Omron CX-Programmer project NewProject (CX-Programmer 9.75)

# PLC NewPLC1: CP2E-N N

## Global symbols (name address type ; comment)
0 CHANNEL  ; VIN1
0.00 BOOL  ; TIMER
0.01 BOOL  ; Auto
0.03 BOOL  ; Manual
1 CHANNEL  ; VIN1
100.01 BOOL  ; Tes
100.03 BOOL  ; 3C4
102 CHANNEL  ; INPUT 1 and 2 ACTIVE, AVERAGING, 0-10 V INPUT
103 CHANNEL  ; INPUT 3 AND 4 0-10V
2 CHANNEL  ; VIN1
3 CHANNEL  ; Potensiometer Input
4 CHANNEL  ; VIN3
5 CHANNEL  ; Timer every 500 ms mengambil data sensor
6 CHANNEL  ; VIN3
7 CHANNEL  ; VIN3
D0 CHANNEL  ; POTENTIOMETER
D1 CHANNEL  ; Panas
D10 CHANNEL  ; Parameter Sensor Suhu
D14 CHANNEL  ; Parameter Potentiometer
D151 CHANNEL  ; BIN to FLOAT Sensor Panas Multiply
D152 CHANNEL  ; Regression Multiply
D153 CHANNEL  ; Sensor Panas Float Unbiased
D154 CHANNEL  ; Bias Sensor Panas
D161 CHANNEL  ; Sensor Panas Float Unscaled
D170 CHANNEL  ; Bin to FLOAT Sensor division
D171 CHANNEL  ; BIN to FLOAT TRANSIMTTER DINGIN
D181 CHANNEL  ; Sensor Dingin Float Unscaled
D182 CHANNEL  ; Sensor Dingin Regression
D183 CHANNEL  ; Sensor Dingin no bias
D2 CHANNEL  ; Dingin
D20 CHANNEL  ; Hysterisis Input
D201 CHANNEL  ; DINGIN BIAS
D21 CHANNEL  ; Float Hysterisis Input
D30 CHANNEL  ; Scaled Sensor Dingin
D31 CHANNEL  ; Scaled Sensor Panas
D32 CHANNEL  ; Scaled Potentiometer FLOAT
D33 CHANNEL  ; Sensor Dingin Scaled
D34 CHANNEL  ; Scaled Sensor Panas
D35 CHANNEL  ; in bcd
D41 CHANNEL  ; Set atas
D42 CHANNEL  ; Set bawah
D70 CHANNEL  ; POTENTIOMETER FLOAT DIVIDER
D71 CHANNEL  ; POTENTIOMETER MULTIP FACTOR
D72 CHANNEL  ; POTENTIOMETER REGRESSION
D77 CHANNEL  ; POTENSIOMETER MULTIP FLOAT
D90 CHANNEL  ; UINT SENSOR DINGIN
D91 CHANNEL  ; UINT SENSOR PANAS
D92 CHANNEL  ; UINT POTENTIOMETER
T000 BOOL  ; TIMER
T001 BOOL  ; TIM2
LAMP 101.00 BOOL  ; Peltier
PELTIER 100.02 BOOL  ; 3C5
Switch 0.00 BOOL

## Program NewProgram1 (cyclic task 0)

### Section Initiation_and_Moving_Var

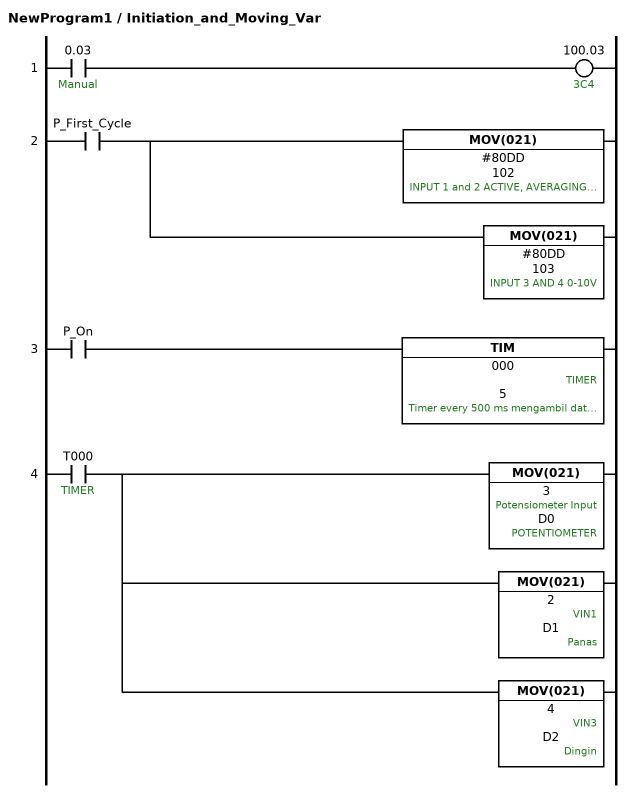
; rung 1
LD 0.03  ; Manual
OUT 100.03  ; 3C4
; rung 2
LD P_First_Cycle
MOV(021) #80DD 102  ; INPUT 1 and 2 ACTIVE, AVERAGING, 0-10 V INPUT
MOV(021) #80DD 103  ; INPUT 3 AND 4 0-10V
; rung 3
LD P_On
TIM 000 5  ; Timer every 500 ms mengambil data sensor, TIMER
; rung 4
LD T000  ; TIMER
MOV(021) 3 D0  ; Potensiometer Input, POTENTIOMETER
MOV(021) 2 D1  ; VIN1, Panas
MOV(021) 4 D2  ; VIN3, Dingin

### Section Scaling

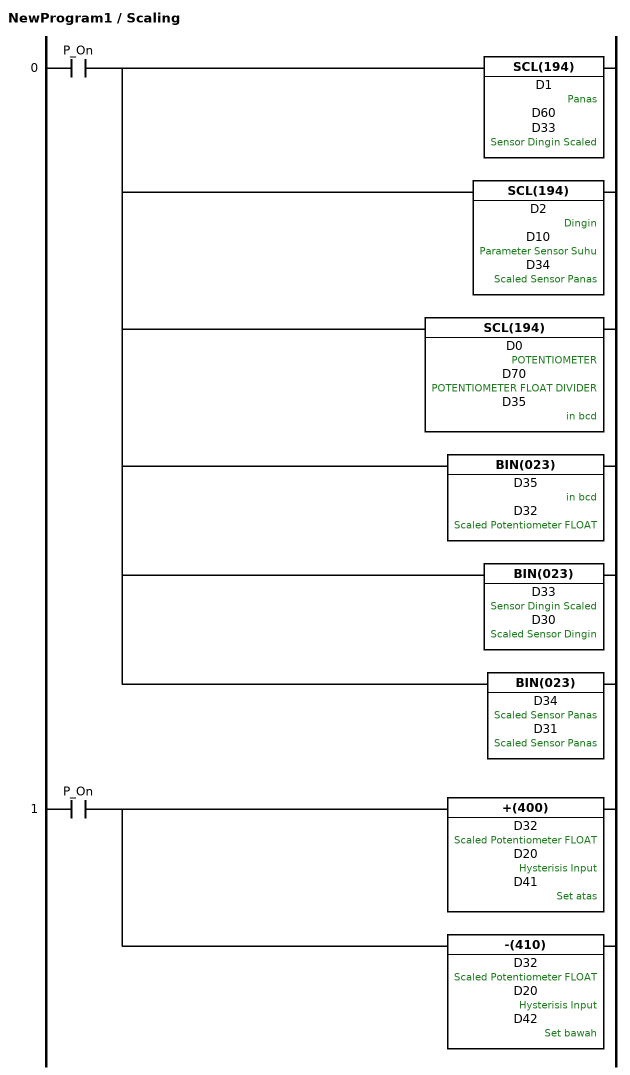
; rung 0
LD P_On
SCL(194) D1 D60 D33  ; Panas, Sensor Dingin Scaled
SCL(194) D2 D10 D34  ; Dingin, Parameter Sensor Suhu, Scaled Sensor Panas
SCL(194) D0 D70 D35  ; POTENTIOMETER, POTENTIOMETER FLOAT DIVIDER, in bcd
BIN(023) D35 D32  ; in bcd, Scaled Potentiometer FLOAT
BIN(023) D33 D30  ; Sensor Dingin Scaled, Scaled Sensor Dingin
BIN(023) D34 D31  ; Scaled Sensor Panas
; rung 1
LD P_On
+(400) D32 D20 D41  ; Scaled Potentiometer FLOAT, Hysterisis Input, Set atas
-(410) D32 D20 D42  ; Scaled Potentiometer FLOAT, Hysterisis Input, Set bawah

### Section Control

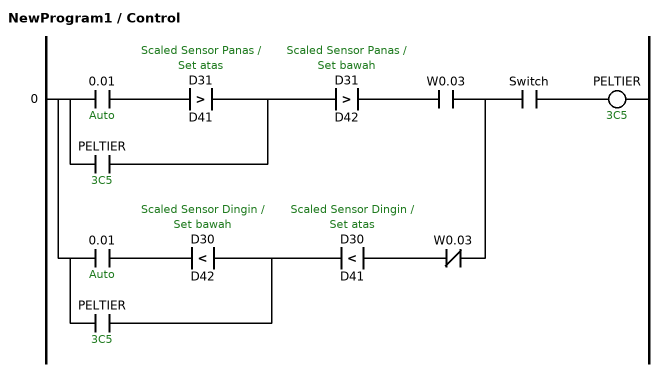
; rung 0
LD 0.01  ; Auto
AND>(320) D31 D41  ; Scaled Sensor Panas, Set atas
OR PELTIER  ; 3C5
AND>(320) D31 D42  ; Scaled Sensor Panas, Set bawah
AND W0.03
LD 0.01  ; Auto
AND<(310) D30 D42  ; Scaled Sensor Dingin, Set bawah
OR PELTIER  ; 3C5
AND<(310) D30 D41  ; Scaled Sensor Dingin, Set atas
ANDNOT W0.03
ORLD
AND Switch
OUT PELTIER  ; 3C5

### Section nyimpen

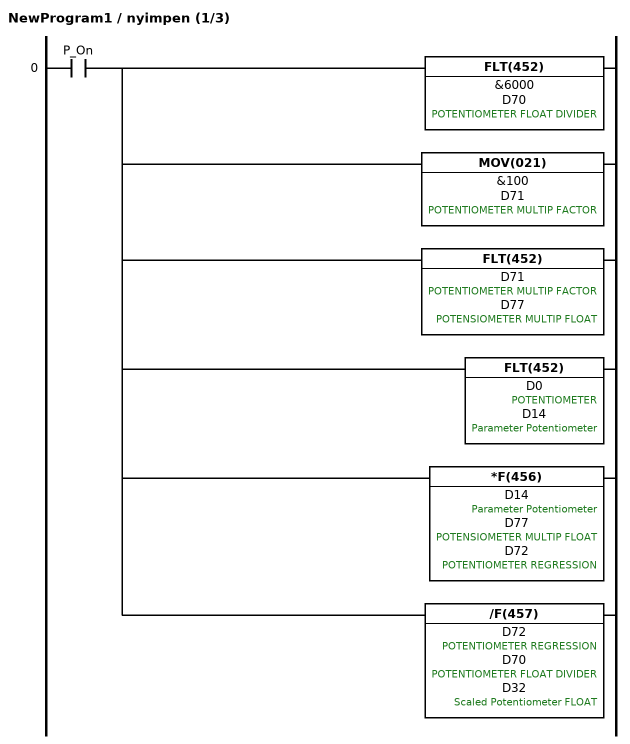
; rung 0
LD P_On
FLT(452) &6000 D70  ; POTENTIOMETER FLOAT DIVIDER
MOV(021) &100 D71  ; POTENTIOMETER MULTIP FACTOR
FLT(452) D71 D77  ; POTENTIOMETER MULTIP FACTOR, POTENSIOMETER MULTIP FLOAT
FLT(452) D0 D14  ; POTENTIOMETER, Parameter Potentiometer
*F(456) D14 D77 D72  ; Parameter Potentiometer, POTENSIOMETER MULTIP FLOAT, POTENTIOMETER REGRESSION
/F(457) D72 D70 D32  ; POTENTIOMETER REGRESSION, POTENTIOMETER FLOAT DIVIDER, Scaled Potentiometer FLOAT

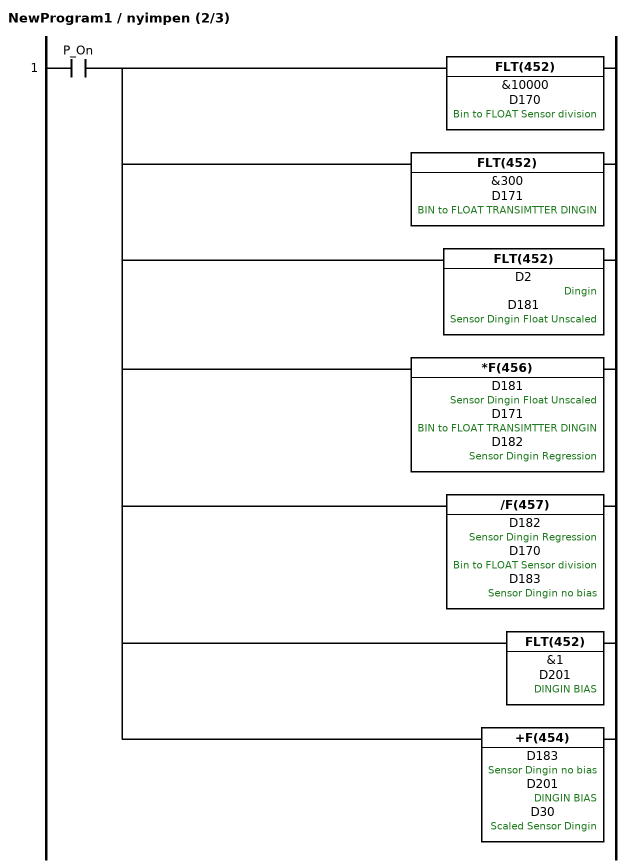
; rung 1
LD P_On
FLT(452) &10000 D170  ; Bin to FLOAT Sensor division
FLT(452) &300 D171  ; BIN to FLOAT TRANSIMTTER DINGIN
FLT(452) D2 D181  ; Dingin, Sensor Dingin Float Unscaled
*F(456) D181 D171 D182  ; Sensor Dingin Float Unscaled, BIN to FLOAT TRANSIMTTER DINGIN, Sensor Dingin Regression
/F(457) D182 D170 D183  ; Sensor Dingin Regression, Bin to FLOAT Sensor division, Sensor Dingin no bias
FLT(452) &1 D201  ; DINGIN BIAS
+F(454) D183 D201 D30  ; Sensor Dingin no bias, DINGIN BIAS, Scaled Sensor Dingin

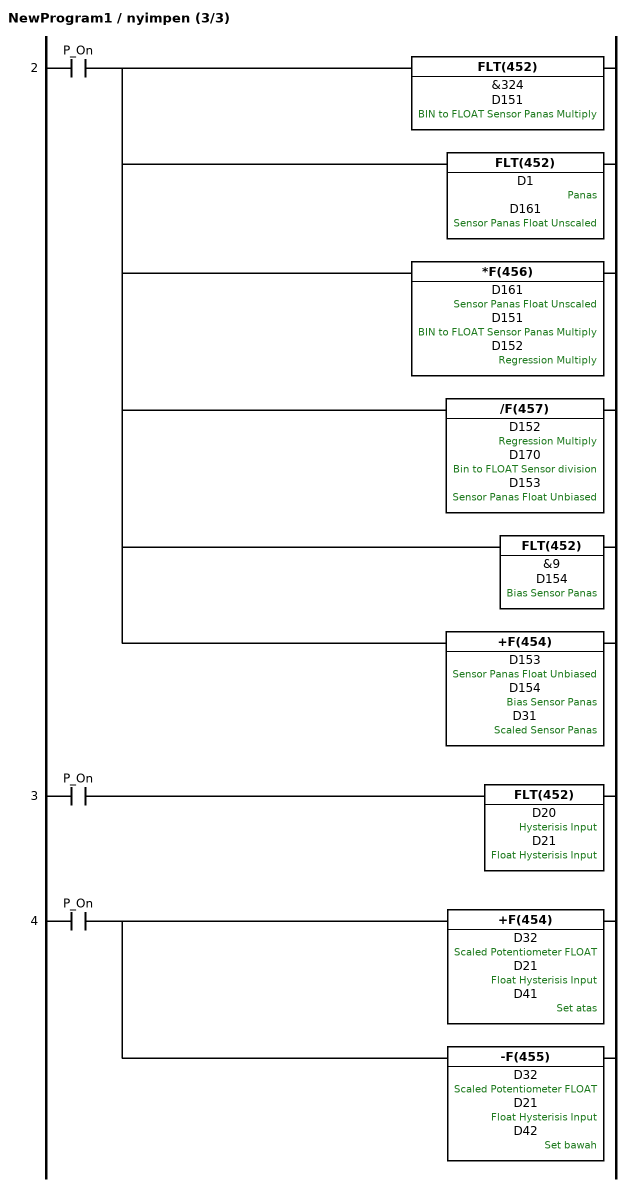
; rung 2
LD P_On
FLT(452) &324 D151  ; BIN to FLOAT Sensor Panas Multiply
FLT(452) D1 D161  ; Panas, Sensor Panas Float Unscaled
*F(456) D161 D151 D152  ; Sensor Panas Float Unscaled, BIN to FLOAT Sensor Panas Multiply, Regression Multiply
/F(457) D152 D170 D153  ; Regression Multiply, Bin to FLOAT Sensor division, Sensor Panas Float Unbiased
FLT(452) &9 D154  ; Bias Sensor Panas
+F(454) D153 D154 D31  ; Sensor Panas Float Unbiased, Bias Sensor Panas, Scaled Sensor Panas
; rung 3
LD P_On
FLT(452) D20 D21  ; Hysterisis Input, Float Hysterisis Input
; rung 4
LD P_On
+F(454) D32 D21 D41  ; Scaled Potentiometer FLOAT, Float Hysterisis Input, Set atas
-F(455) D32 D21 D42  ; Scaled Potentiometer FLOAT, Float Hysterisis Input, Set bawah

### Section END
; rung 0
END(001)